// SIMATIC S7-200 SMART project (STEP 7-Micro/WIN SMART), CPU SR40

ORGANIZATION_BLOCK MAIN:OB1
TITLE=程序注释
BEGIN
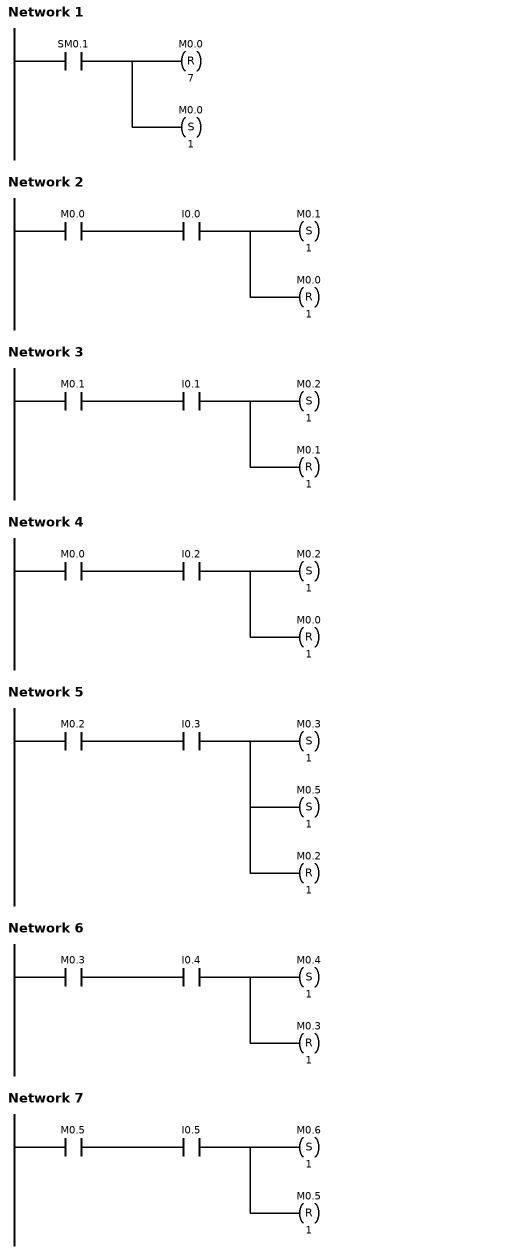
Network 1
LD     SM0.1
R      M0.0, 7
S      M0.0, 1
Network 2
LD     M0.0
A      I0.0
S      M0.1, 1
R      M0.0, 1
Network 3
LD     M0.1
A      I0.1
S      M0.2, 1
R      M0.1, 1
Network 4
LD     M0.0
A      I0.2
S      M0.2, 1
R      M0.0, 1
Network 5
LD     M0.2
A      I0.3
S      M0.3, 1
S      M0.5, 1
R      M0.2, 1
Network 6
LD     M0.3
A      I0.4
S      M0.4, 1
R      M0.3, 1
Network 7
LD     M0.5
A      I0.5
S      M0.6, 1
R      M0.5, 1
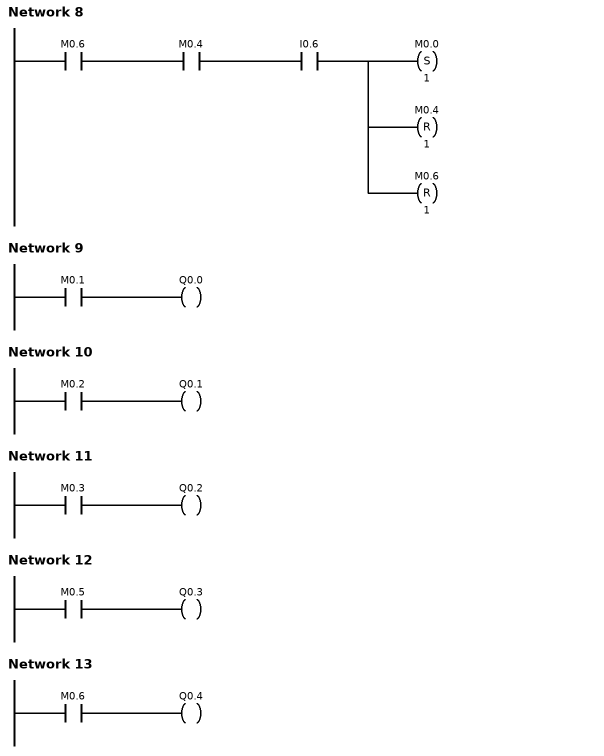
Network 8
LD     M0.6
A      M0.4
A      I0.6
S      M0.0, 1
R      M0.4, 1
R      M0.6, 1
Network 9
LD     M0.1
=      Q0.0
Network 10
LD     M0.2
=      Q0.1
Network 11
LD     M0.3
=      Q0.2
Network 12
LD     M0.5
=      Q0.3
Network 13
LD     M0.6
=      Q0.4
END_ORGANIZATION_BLOCK
